PROGRAM MAIN_HMI
VAR
END_VAR

END_PROGRAM

(* stored: Version 1.1.0.1, ProductVersion 3.1.4024.15
   POU MAIN_HMI: Id {3c91d346-e8aa-4b63-90ca-940de5bd825a}, SpecialFunc None *)
